{attribute 'linkalways'}
{attribute 'hide_all_locals'}
FUNCTION_BLOCK ValueDateRead EXTENDS ValueBase IMPLEMENTS ValueRead
VAR
	thisValue : DATE;
END_VAR

{attribute 'call_after_global_init_slot' := '1'}
{attribute 'call_after_online_change_slot' := '1'}
METHOD PROTECTED GetThisAnyType
VAR_INPUT
END_VAR
thisAnyType := ToAnyType(thisValue);
END_METHOD

METHOD GetAsType : BOOL
VAR_INPUT
	destination : __SYSTEM.AnyType;
END_VAR
GetAsType := ConvertAnyType(thisAnyType, destination);
END_METHOD

METHOD GetAsString : T_MaxString
VAR_INPUT
END_VAR
GetAsString := DATE_TO_STRING(thisValue);
END_METHOD

METHOD Get : BOOL
VAR_INPUT
	destination : ANY;
END_VAR
Get := ConvertAnyType(thisAnyType, destination);
END_METHOD

METHOD FB_init : BOOL
VAR_INPUT
	bInitRetains : BOOL; // if TRUE, the retain variables are initialized (warm start / cold start)
	bInCopyCode : BOOL;  // if TRUE, the instance afterwards gets moved into the copy code (online change)
END_VAR
_ValueType := __SYSTEM.TYPE_CLASS.TYPE_DATE;
END_METHOD

{attribute 'monitoring' := 'call'}
PROPERTY Value : DATE
GET
Value := thisValue;
END_GET
END_PROPERTY

END_FUNCTION_BLOCK

(* stored: Version 1.1.0.1
   POU ValueDateRead: Id {531db2cf-6e68-4683-9aaf-1e8298e750f1}, SpecialFunc None
   Method GetThisAnyType: Id {8f3e7c5d-df98-44cf-a257-cec3247ec359}
   Method GetAsType: Id {9b93afbc-475e-4d5a-a178-c05ac05ba328}
   Method GetAsString: Id {8ead77d6-aea8-4fbe-8ad3-2a49c62f1d22}
   Method Get: Id {402650bc-dd8e-4a00-b4e1-85e77a67910b}
   Method FB_init: Id {af769c3c-619a-4a37-a48d-1f5ca604f894}
   Property Value: Id {94ae888e-85ea-4aab-85fd-3d214ad5d176}
   Get Get: Id {2765b59a-7824-45c0-84b9-2b2f9e9b149b} *)
